(* CODESYS project Group6_Assigment_2_Elevators.export

Project tree, tasks and I/O mapping:
  control/
    function block DoorCtrl [SFC]
    program ElevatorControl [LD]
    program main [ST]
*)

// control/DoorCtrl
FUNCTION_BLOCK DoorCtrl
VAR_INPUT
	open: BOOL;
	precondtion: BOOL;
	forceClose: BOOL;
	openedSensor: BOOL;
	closedSensor: BOOL;
END_VAR
VAR_OUTPUT
	executing: BOOL;
	closed: BOOL;
	openControl: BOOL;
END_VAR
VAR
END_VAR

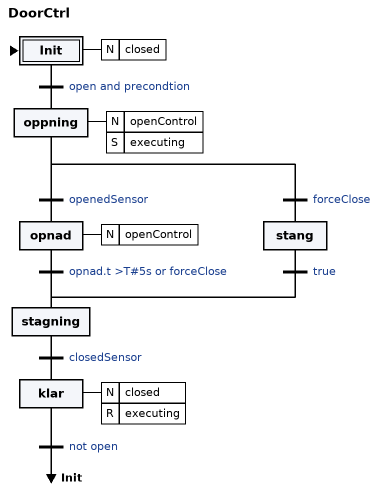
INITIAL_STEP Init:
    closed(N);
END_STEP
TRANSITION FROM Init TO oppning
    := open and precondtion;
END_TRANSITION
STEP oppning:
    openControl(N);
    executing(S);
END_STEP
TRANSITION FROM oppning TO opnad
    := openedSensor;
END_TRANSITION
STEP opnad:
    openControl(N);
END_STEP
TRANSITION FROM opnad TO stagning
    := opnad.t >T#5s or forceClose;
END_TRANSITION
TRANSITION FROM oppning TO stang
    := forceClose;
END_TRANSITION
STEP stang:
END_STEP
TRANSITION FROM stang TO stagning
    := true;
END_TRANSITION
STEP stagning:
END_STEP
TRANSITION FROM stagning TO klar
    := closedSensor;
END_TRANSITION
STEP klar:
    closed(N);
    executing(R);
END_STEP
TRANSITION FROM klar TO Init
    := not open;
END_TRANSITION

END_FUNCTION_BLOCK

// control/ElevatorControl
PROGRAM ElevatorControl
VAR
	up: BOOL;
	down: BOOL;
	DoorIsOpen: BOOL;
	requestF1: BOOL;
	requestF2: BOOL;
	requestF3: BOOL;
	requestF4: BOOL := TRUE;
	DoorsF1: DoorCtrl;
	DoorsF2: DoorCtrl;
	DoorsF3: DoorCtrl;
	DoorsF4: DoorCtrl;
END_VAR

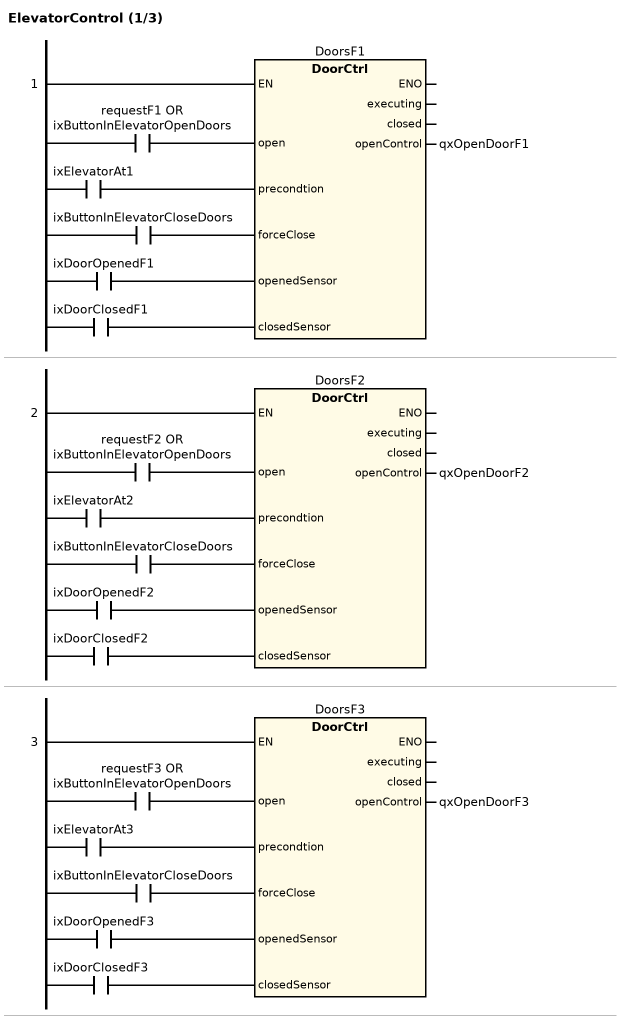
// NETWORK 1
DoorsF1(
    open := requestF1 OR ixButtonInElevatorOpenDoors,
    precondtion := ixElevatorAt1,
    forceClose := ixButtonInElevatorCloseDoors,
    openedSensor := ixDoorOpenedF1,
    closedSensor := ixDoorClosedF1,
    openControl => qxOpenDoorF1); // DoorCtrl

// NETWORK 2
DoorsF2(
    open := requestF2 OR ixButtonInElevatorOpenDoors,
    precondtion := ixElevatorAt2,
    forceClose := ixButtonInElevatorCloseDoors,
    openedSensor := ixDoorOpenedF2,
    closedSensor := ixDoorClosedF2,
    openControl => qxOpenDoorF2); // DoorCtrl

// NETWORK 3
DoorsF3(
    open := requestF3 OR ixButtonInElevatorOpenDoors,
    precondtion := ixElevatorAt3,
    forceClose := ixButtonInElevatorCloseDoors,
    openedSensor := ixDoorOpenedF3,
    closedSensor := ixDoorClosedF3,
    openControl => qxOpenDoorF3); // DoorCtrl

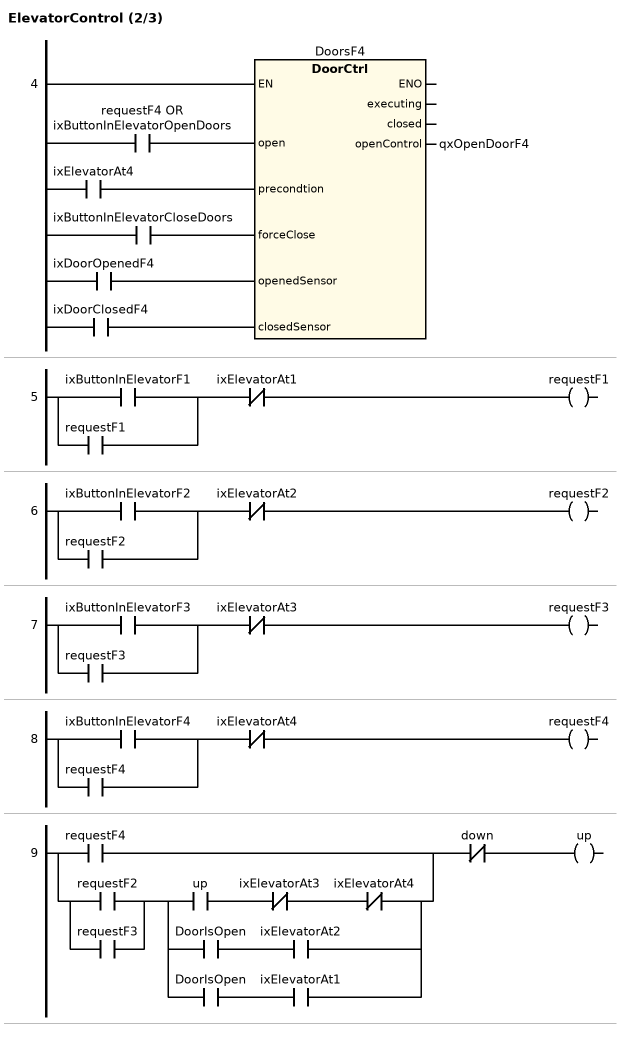
// NETWORK 4
DoorsF4(
    open := requestF4 OR ixButtonInElevatorOpenDoors,
    precondtion := ixElevatorAt4,
    forceClose := ixButtonInElevatorCloseDoors,
    openedSensor := ixDoorOpenedF4,
    closedSensor := ixDoorClosedF4,
    openControl => qxOpenDoorF4); // DoorCtrl

// NETWORK 5
requestF1 := (ixButtonInElevatorF1 OR requestF1) AND NOT ixElevatorAt1;

// NETWORK 6
requestF2 := (ixButtonInElevatorF2 OR requestF2) AND NOT ixElevatorAt2;

// NETWORK 7
requestF3 := (ixButtonInElevatorF3 OR requestF3) AND NOT ixElevatorAt3;

// NETWORK 8
requestF4 := (ixButtonInElevatorF4 OR requestF4) AND NOT ixElevatorAt4;

// NETWORK 9
up := (requestF4 OR (requestF2 OR requestF3) AND (up AND NOT ixElevatorAt3 AND NOT ixElevatorAt4 OR DoorIsOpen AND ixElevatorAt2 OR DoorIsOpen AND ixElevatorAt1)) AND NOT down;

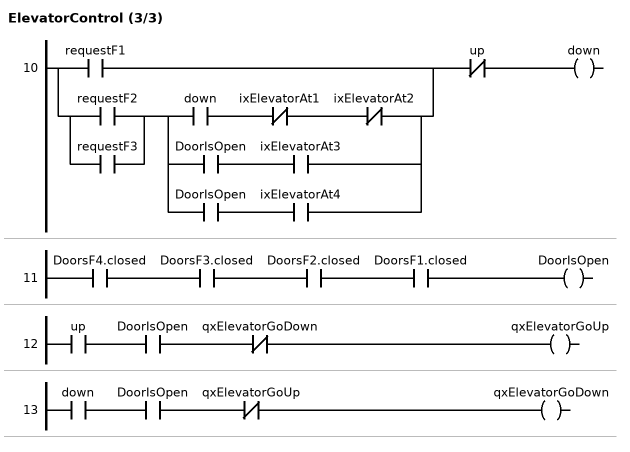
// NETWORK 10
down := (requestF1 OR (requestF2 OR requestF3) AND (down AND NOT ixElevatorAt1 AND NOT ixElevatorAt2 OR DoorIsOpen AND ixElevatorAt3 OR DoorIsOpen AND ixElevatorAt4)) AND NOT up;

// NETWORK 11
DoorIsOpen := DoorsF4.closed AND DoorsF3.closed AND DoorsF2.closed AND DoorsF1.closed;

// NETWORK 12
qxElevatorGoUp := up AND DoorIsOpen AND NOT qxElevatorGoDown;

// NETWORK 13
qxElevatorGoDown := down AND DoorIsOpen AND NOT qxElevatorGoUp;

END_PROGRAM

// control/main
PROGRAM main
VAR
END_VAR

ElevatorControl();

END_PROGRAM
